{attribute 'qualified_only'}
VAR_GLOBAL
	Inicio:BOOL;
	PesoMaxConte:REAL;
	Dosis:REAL;
	Tinyeccion:DINT;
	PesoBatch:REAL;
	Tolerancia:REAL;
	Pausa:BOOL;		
	Error:REAL;
	ContLleno:BOOL;	
	CantPesadas:INT;
	PesoCalibracion:REAL;
	Muestra1_Ok:BOOL;
	Finalizado:BOOL;
	PesoPromedio6:REAL;
	
END_VAR

(* stored: Version 1.1.0.1, ProductVersion 3.1.4024.12
   GVL HMIcalP2: Id {672f6fde-ac02-4614-9ef6-e73b7ba72741} *)
